INTERFACE INTERNAL I_Strb

METHOD Append : I_Strb;
VAR_INPUT
	sToAdd		: Str;
END_VAR
END_METHOD

METHOD FindFirstAfter 	: I_Strb;
VAR_INPUT
	sToFind			: Str;
	nPosition		: INT := 1;
END_VAR
VAR_OUTPUT
	nStart			: INT;
	nEnd			: INT;
END_VAR
END_METHOD

METHOD FindLastBefore 	: I_Strb;
VAR_INPUT
	sToFind			: Str;
	nPosition		: INT := 256;
END_VAR
VAR_OUTPUT
	nStart			: INT;
	nEnd			: INT;
END_VAR
END_METHOD

METHOD HasAfter : BOOL
VAR_INPUT
	sToFind		: Str;
	nPosition	: INT := 0;
END_VAR
VAR_OUTPUT
	nStart			: INT;
	nEnd			: INT;
END_VAR
END_METHOD

METHOD HasBefore : BOOL
VAR_INPUT
	sToFind		: Str;
	nPosition	: INT := 256;
END_VAR
VAR_OUTPUT
	nStart			: INT;
	nEnd			: INT;
END_VAR
END_METHOD

METHOD Inject : I_Strb
VAR_INPUT
	nPosition	: INT;
	sToInject	: Str;
END_VAR
END_METHOD

METHOD IsEmpty : BOOL
VAR_INPUT
END_VAR
END_METHOD

METHOD Length : INT;
VAR_INPUT
END_VAR
END_METHOD

METHOD Prepend : I_Strb;
VAR_INPUT
	sToAdd		: Str;
END_VAR
END_METHOD

METHOD Read : Str;
VAR_INPUT
END_VAR
END_METHOD

METHOD Remove : I_Strb;
VAR_INPUT
	nLength		: INT;
	nPosition	: INT;
END_VAR
END_METHOD

METHOD Set : I_Strb;
VAR_INPUT
	sLiteral	: Str;
END_VAR
END_METHOD

METHOD Slice : I_Strb
VAR_INPUT
	nPosition	: INT;
	nLength		: INT;
END_VAR
VAR_OUTPUT
	sSlice			: Strb;
END_VAR
END_METHOD

METHOD Split : I_Strb;
VAR_INPUT
	nPosition	: INT;
END_VAR
VAR_OUTPUT
	sLeft		: Strb;
	sRight		: Strb;
END_VAR
END_METHOD

END_INTERFACE

(* stored: Version 1.1.0.1
   Itf I_Strb: Id {5d2bb437-ad4f-4366-b0e4-2dbdfc640151}
   Method Append: Id {4b270f4c-6096-4a21-88a7-6f8529989adb}
   Method FindFirstAfter: Id {7a706f6c-b1a7-48a1-a3fe-17b02c7f77da}
   Method FindLastBefore: Id {96548900-e520-4415-b8cc-5a51395d457b}
   Method HasAfter: Id {4ec10599-5406-42a1-8292-64d483624fff}
   Method HasBefore: Id {b7b8682e-6d22-48e1-8967-184f637122bb}
   Method Inject: Id {6518b446-2be2-41a8-94b7-37ecc15088f9}
   Method IsEmpty: Id {d4bb4e76-ce2e-431a-a0d0-037174ed5ed3}
   Method Length: Id {f51afbf3-b882-45dc-9e57-0b2b139d385f}
   Method Prepend: Id {6ecd6cc1-d0f0-436f-af5d-f38c0c477991}
   Method Read: Id {5fc32b24-95f4-40aa-9417-d850d57aa806}
   Method Remove: Id {4c25a438-0f2e-4285-882b-3038bdf8236f}
   Method Set: Id {39dce832-4c61-4887-a2a5-655777ad4758}
   Method Slice: Id {b0ce04e8-82ba-4ad1-9c5b-9ec7358e16f5}
   Method Split: Id {6b5516c8-cca4-4cba-9a64-2a6f94350f39} *)
